(* Logix 5000 project; controller R1USB70001_CWRU_Scenario_Gen_20111116 vendor 1 type 14 code 54 rev 19.11; software revision 19.01; part 4 of 6 *)
(* tags used below, declared in another part *)
   EditScenarioPv : EditScenarioPv;
   HMIPv : HMIPv;
   CL_LP_B1_SG : ALIAS FOR ACNR_CP_SG_N5:1:O.1;
   CL_LP_ML_SG : ALIAS FOR ACNR_CP_SG_N5:1:O.0;
   EditScenario : EditScenarioPub;
   HMI : HMIPub;
   HMI_Intfc_Write_Buffer : DINT[20];
   RL_LP_B1_SG : ALIAS FOR ACNR_RP_SG_N4:1:O.1;
   RL_LP_B2_SG : ALIAS FOR ACNR_RP_SG_N4:2:O.4;
   RL_LP_B3_SG : ALIAS FOR ACNR_RP_SG_N4:3:O.7;
   RL_LP_B4_SG : ALIAS FOR ACNR_RP_SG_N4:5:O.2;
   RL_LP_ML_SG : ALIAS FOR ACNR_RP_SG_N4:1:O.0;
   Scenario : Scenario_Def[100];
(* MainProgram, continued *)

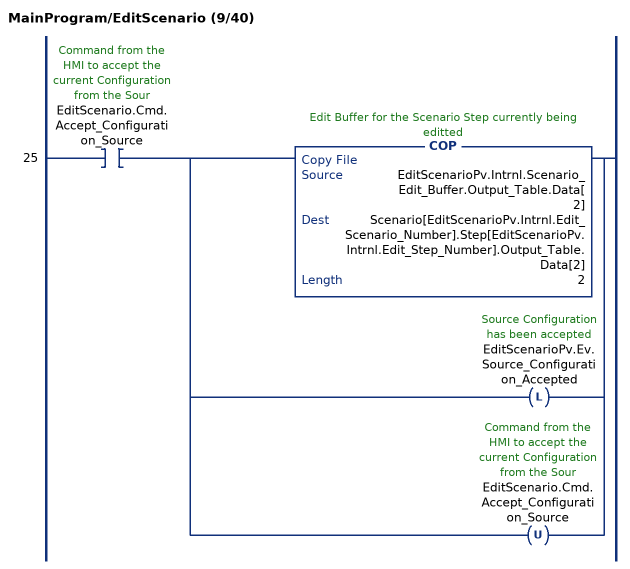
   25: XIC(EditScenario.Cmd.Accept_Configuration_Source)[COP(EditScenarioPv.Intrnl.Scenario_Edit_Buffer.Output_Table.Data[2],Scenario[EditScenarioPv.Intrnl.Edit_Scenario_Number].Step[EditScenarioPv.Intrnl.Edit_Step_Number].Output_Table.Data[2],2) ,OTL(EditScenarioPv.Ev.Source_Configuration_Accepted) ,OTU(EditScenario.Cmd.Accept_Configuration_Source) ];
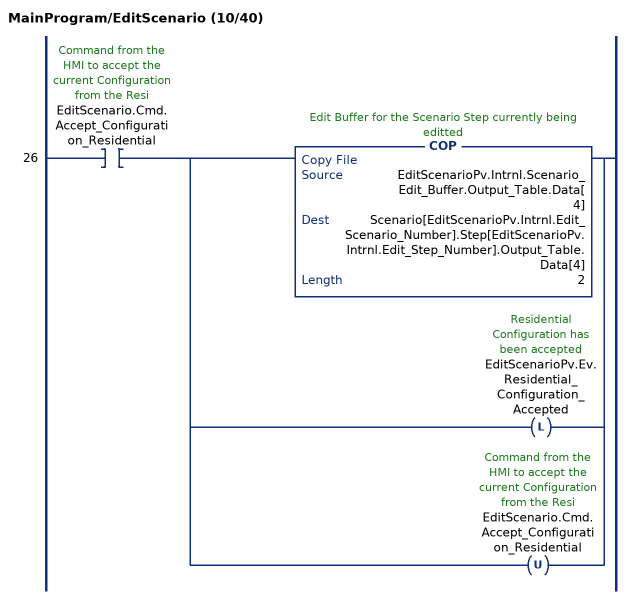
   26: XIC(EditScenario.Cmd.Accept_Configuration_Residential)[COP(EditScenarioPv.Intrnl.Scenario_Edit_Buffer.Output_Table.Data[4],Scenario[EditScenarioPv.Intrnl.Edit_Scenario_Number].Step[EditScenarioPv.Intrnl.Edit_Step_Number].Output_Table.Data[4],2) ,OTL(EditScenarioPv.Ev.Residential_Configuration_Accepted) ,OTU(EditScenario.Cmd.Accept_Configuration_Residential) ];
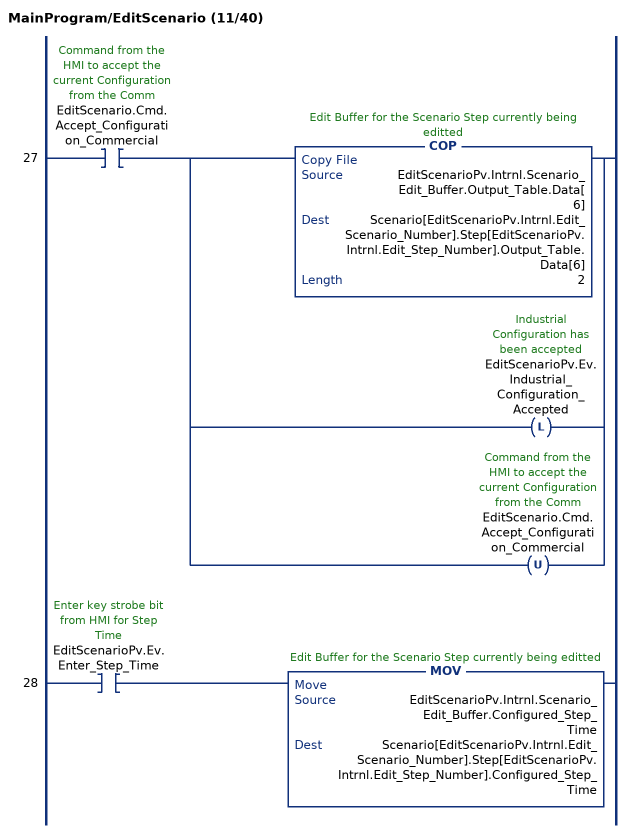
   27: XIC(EditScenario.Cmd.Accept_Configuration_Commercial)[COP(EditScenarioPv.Intrnl.Scenario_Edit_Buffer.Output_Table.Data[6],Scenario[EditScenarioPv.Intrnl.Edit_Scenario_Number].Step[EditScenarioPv.Intrnl.Edit_Step_Number].Output_Table.Data[6],2) ,OTL(EditScenarioPv.Ev.Industrial_Configuration_Accepted) ,OTU(EditScenario.Cmd.Accept_Configuration_Commercial) ];
   28: XIC(EditScenarioPv.Ev.Enter_Step_Time)MOV(EditScenarioPv.Intrnl.Scenario_Edit_Buffer.Configured_Step_Time,Scenario[EditScenarioPv.Intrnl.Edit_Scenario_Number].Step[EditScenarioPv.Intrnl.Edit_Step_Number].Configured_Step_Time);
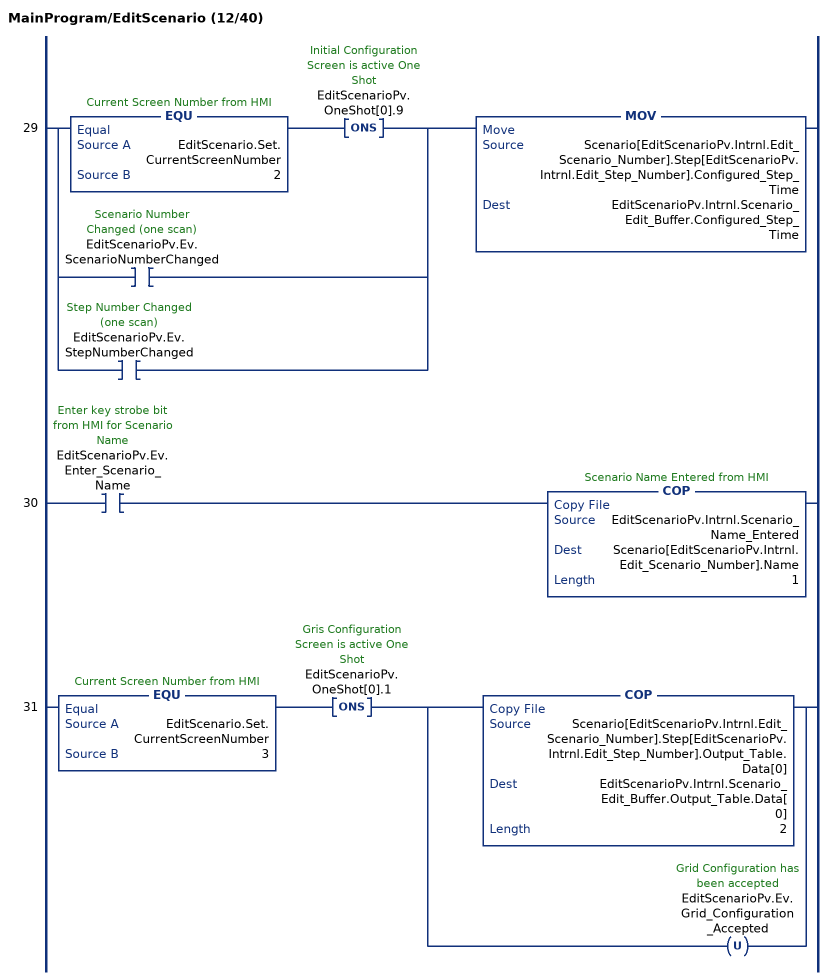
   29: [EQU(EditScenario.Set.CurrentScreenNumber,2) ONS(EditScenarioPv.OneShot[0].9) ,XIC(EditScenarioPv.Ev.ScenarioNumberChanged) ,XIC(EditScenarioPv.Ev.StepNumberChanged) ]MOV(Scenario[EditScenarioPv.Intrnl.Edit_Scenario_Number].Step[EditScenarioPv.Intrnl.Edit_Step_Number].Configured_Step_Time,EditScenarioPv.Intrnl.Scenario_Edit_Buffer.Configured_Step_Time);
   30: XIC(EditScenarioPv.Ev.Enter_Scenario_Name)COP(EditScenarioPv.Intrnl.Scenario_Name_Entered,Scenario[EditScenarioPv.Intrnl.Edit_Scenario_Number].Name,1);
   31: EQU(EditScenario.Set.CurrentScreenNumber,3)ONS(EditScenarioPv.OneShot[0].1)[COP(Scenario[EditScenarioPv.Intrnl.Edit_Scenario_Number].Step[EditScenarioPv.Intrnl.Edit_Step_Number].Output_Table.Data[0],EditScenarioPv.Intrnl.Scenario_Edit_Buffer.Output_Table.Data[0],2) ,OTU(EditScenarioPv.Ev.Grid_Configuration_Accepted) ];
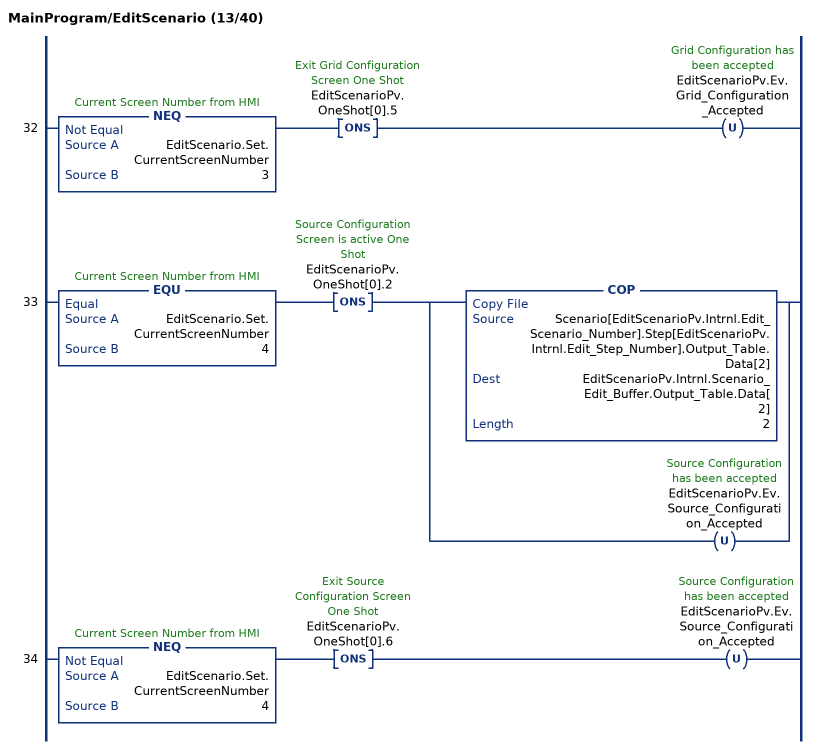
   32: NEQ(EditScenario.Set.CurrentScreenNumber,3)ONS(EditScenarioPv.OneShot[0].5)OTU(EditScenarioPv.Ev.Grid_Configuration_Accepted);
   33: EQU(EditScenario.Set.CurrentScreenNumber,4)ONS(EditScenarioPv.OneShot[0].2)[COP(Scenario[EditScenarioPv.Intrnl.Edit_Scenario_Number].Step[EditScenarioPv.Intrnl.Edit_Step_Number].Output_Table.Data[2],EditScenarioPv.Intrnl.Scenario_Edit_Buffer.Output_Table.Data[2],2) ,OTU(EditScenarioPv.Ev.Source_Configuration_Accepted) ];
   34: NEQ(EditScenario.Set.CurrentScreenNumber,4)ONS(EditScenarioPv.OneShot[0].6)OTU(EditScenarioPv.Ev.Source_Configuration_Accepted);
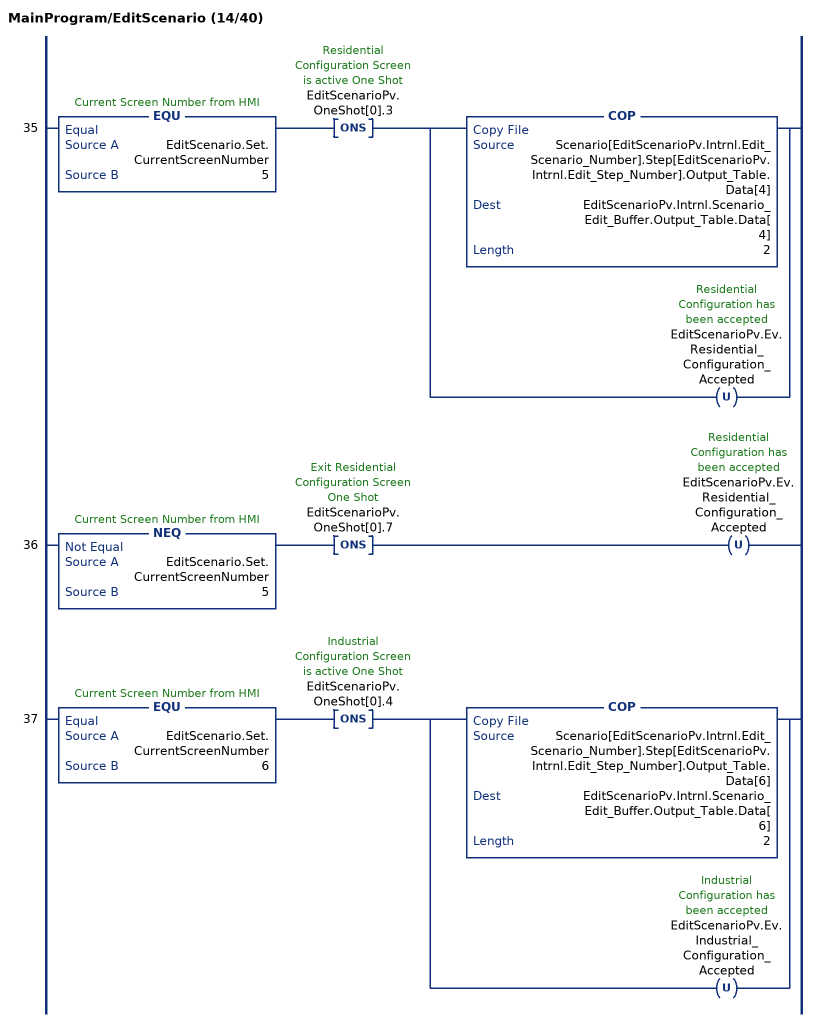
   35: EQU(EditScenario.Set.CurrentScreenNumber,5)ONS(EditScenarioPv.OneShot[0].3)[COP(Scenario[EditScenarioPv.Intrnl.Edit_Scenario_Number].Step[EditScenarioPv.Intrnl.Edit_Step_Number].Output_Table.Data[4],EditScenarioPv.Intrnl.Scenario_Edit_Buffer.Output_Table.Data[4],2) ,OTU(EditScenarioPv.Ev.Residential_Configuration_Accepted) ];
   36: NEQ(EditScenario.Set.CurrentScreenNumber,5)ONS(EditScenarioPv.OneShot[0].7)OTU(EditScenarioPv.Ev.Residential_Configuration_Accepted);
   37: EQU(EditScenario.Set.CurrentScreenNumber,6)ONS(EditScenarioPv.OneShot[0].4)[COP(Scenario[EditScenarioPv.Intrnl.Edit_Scenario_Number].Step[EditScenarioPv.Intrnl.Edit_Step_Number].Output_Table.Data[6],EditScenarioPv.Intrnl.Scenario_Edit_Buffer.Output_Table.Data[6],2) ,OTU(EditScenarioPv.Ev.Industrial_Configuration_Accepted) ];
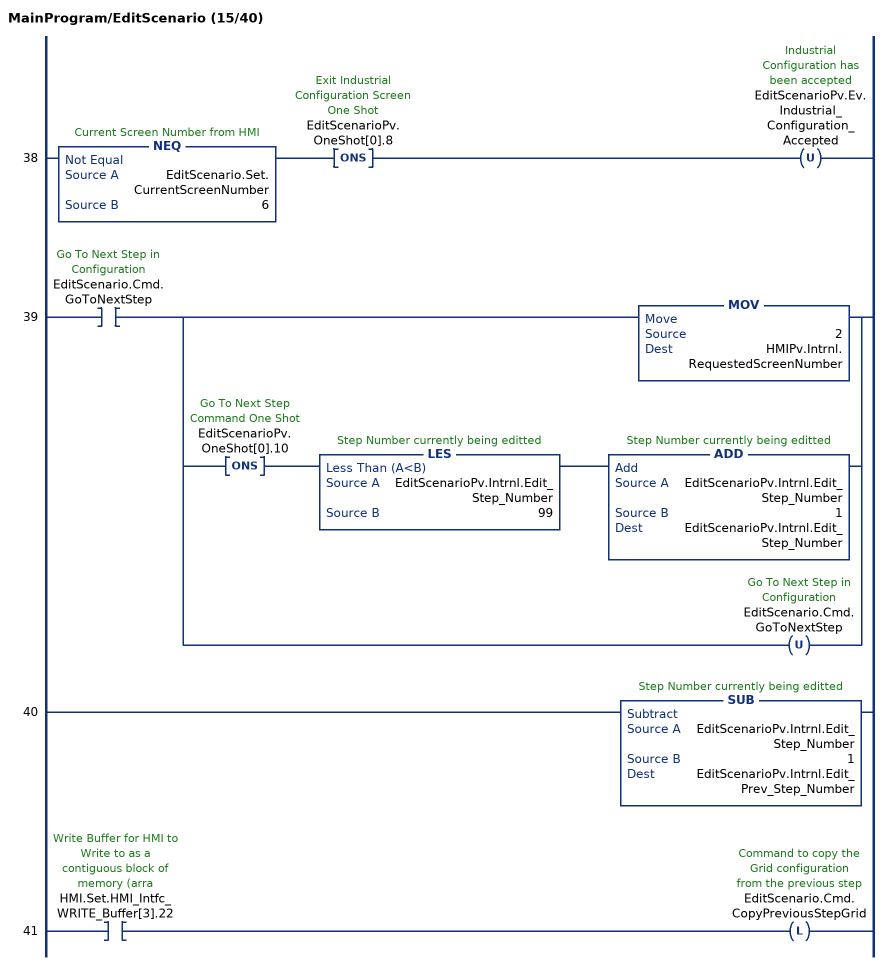
   38: NEQ(EditScenario.Set.CurrentScreenNumber,6)ONS(EditScenarioPv.OneShot[0].8)OTU(EditScenarioPv.Ev.Industrial_Configuration_Accepted);
   39: XIC(EditScenario.Cmd.GoToNextStep)[MOV(2,HMIPv.Intrnl.RequestedScreenNumber) ,ONS(EditScenarioPv.OneShot[0].10) LES(EditScenarioPv.Intrnl.Edit_Step_Number,99) ADD(EditScenarioPv.Intrnl.Edit_Step_Number,1,EditScenarioPv.Intrnl.Edit_Step_Number) ,OTU(EditScenario.Cmd.GoToNextStep) ];
   40: SUB(EditScenarioPv.Intrnl.Edit_Step_Number,1,EditScenarioPv.Intrnl.Edit_Prev_Step_Number);
   41: XIC(HMI.Set.HMI_Intfc_WRITE_Buffer[3].22)OTL(EditScenario.Cmd.CopyPreviousStepGrid);
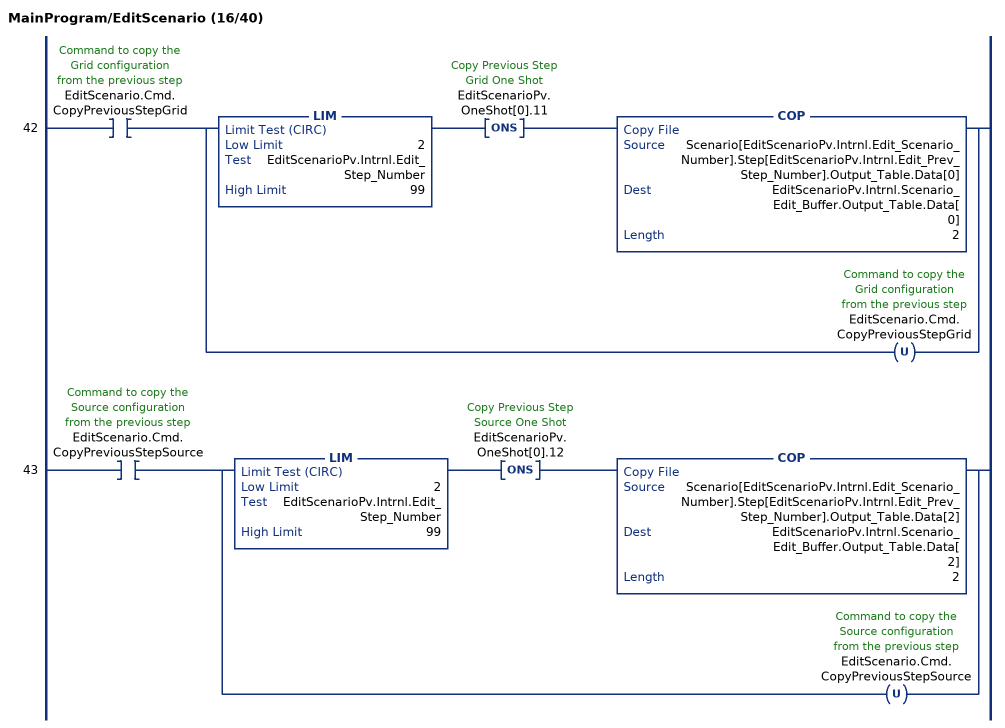
   42: XIC(EditScenario.Cmd.CopyPreviousStepGrid)[LIM(2,EditScenarioPv.Intrnl.Edit_Step_Number,99) ONS(EditScenarioPv.OneShot[0].11) COP(Scenario[EditScenarioPv.Intrnl.Edit_Scenario_Number].Step[EditScenarioPv.Intrnl.Edit_Prev_Step_Number].Output_Table.Data[0],EditScenarioPv.Intrnl.Scenario_Edit_Buffer.Output_Table.Data[0],2) ,OTU(EditScenario.Cmd.CopyPreviousStepGrid) ];
   43: XIC(EditScenario.Cmd.CopyPreviousStepSource)[LIM(2,EditScenarioPv.Intrnl.Edit_Step_Number,99) ONS(EditScenarioPv.OneShot[0].12) COP(Scenario[EditScenarioPv.Intrnl.Edit_Scenario_Number].Step[EditScenarioPv.Intrnl.Edit_Prev_Step_Number].Output_Table.Data[2],EditScenarioPv.Intrnl.Scenario_Edit_Buffer.Output_Table.Data[2],2) ,OTU(EditScenario.Cmd.CopyPreviousStepSource) ];
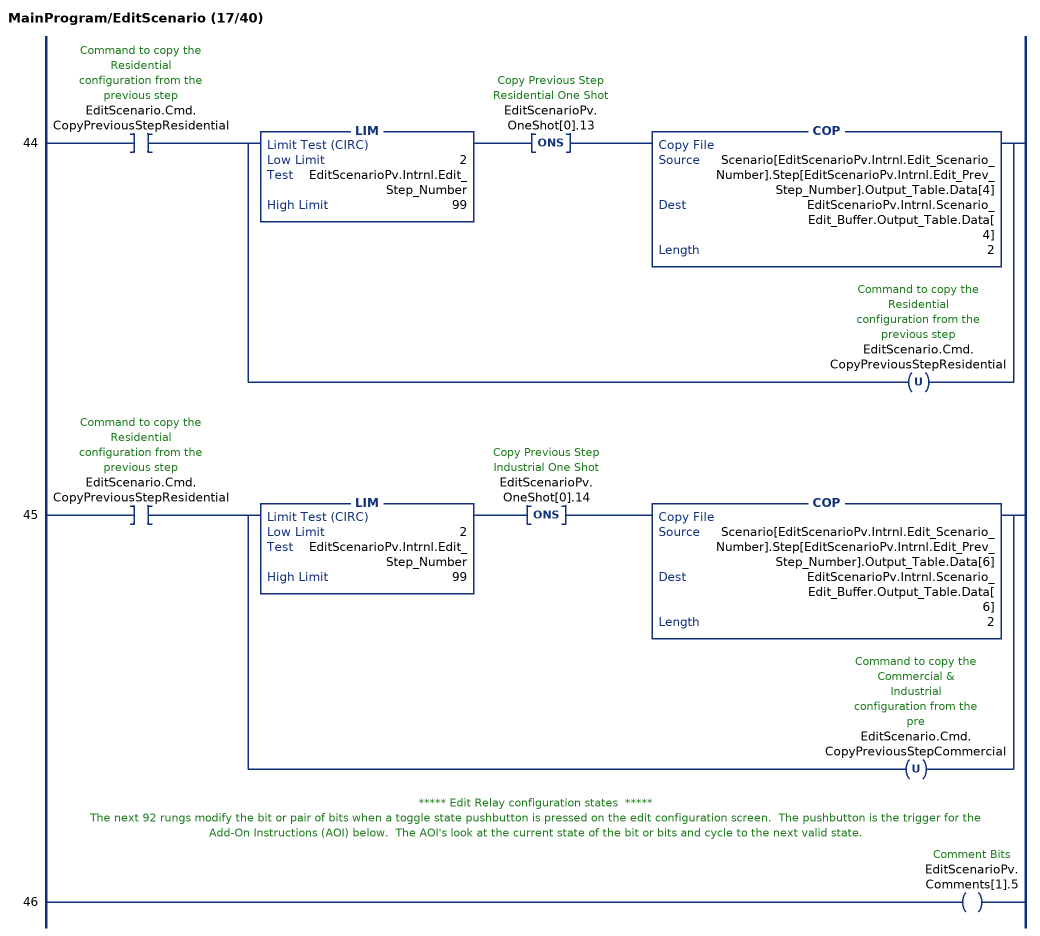
   44: XIC(EditScenario.Cmd.CopyPreviousStepResidential)[LIM(2,EditScenarioPv.Intrnl.Edit_Step_Number,99) ONS(EditScenarioPv.OneShot[0].13) COP(Scenario[EditScenarioPv.Intrnl.Edit_Scenario_Number].Step[EditScenarioPv.Intrnl.Edit_Prev_Step_Number].Output_Table.Data[4],EditScenarioPv.Intrnl.Scenario_Edit_Buffer.Output_Table.Data[4],2) ,OTU(EditScenario.Cmd.CopyPreviousStepResidential) ];
   45: XIC(EditScenario.Cmd.CopyPreviousStepResidential)[LIM(2,EditScenarioPv.Intrnl.Edit_Step_Number,99) ONS(EditScenarioPv.OneShot[0].14) COP(Scenario[EditScenarioPv.Intrnl.Edit_Scenario_Number].Step[EditScenarioPv.Intrnl.Edit_Prev_Step_Number].Output_Table.Data[6],EditScenarioPv.Intrnl.Scenario_Edit_Buffer.Output_Table.Data[6],2) ,OTU(EditScenario.Cmd.CopyPreviousStepCommercial) ];
   // ***** Edit Relay configuration states  *****
   // The next 92 rungs modify the bit or pair of bits when a toggle state pushbutton is pressed on the edit configuration screen.  The pushbutton is the trigger for the Add-On Instructions (AOI) below.  The AOI's look at the current state of the bit or bits and cycle to the next valid state.
   46: OTE(EditScenarioPv.Comments[1].5);
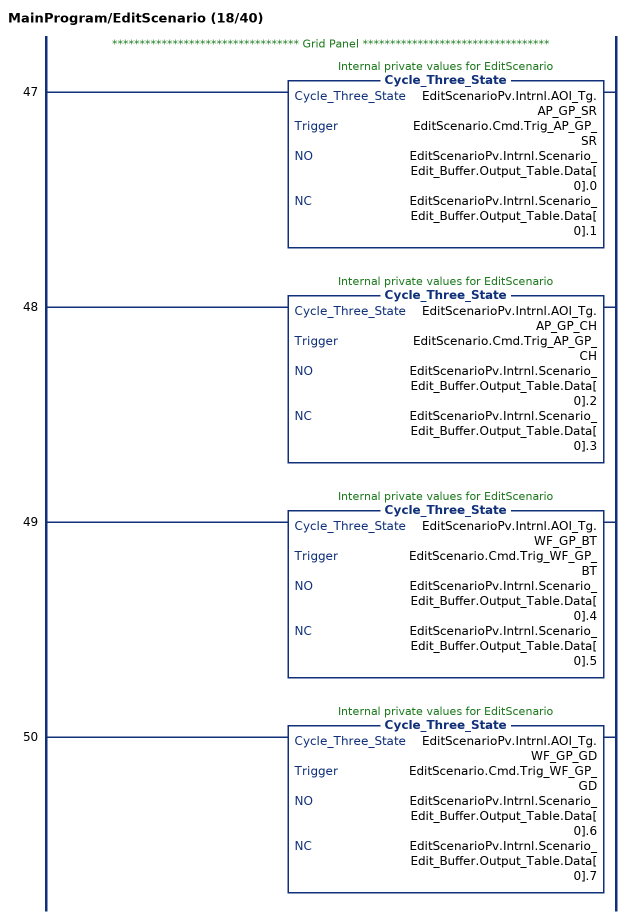
   // ********************************** Grid Panel **********************************
   47: Cycle_Three_State(EditScenarioPv.Intrnl.AOI_Tg.AP_GP_SR,EditScenario.Cmd.Trig_AP_GP_SR,EditScenarioPv.Intrnl.Scenario_Edit_Buffer.Output_Table.Data[0].0,EditScenarioPv.Intrnl.Scenario_Edit_Buffer.Output_Table.Data[0].1);
   48: Cycle_Three_State(EditScenarioPv.Intrnl.AOI_Tg.AP_GP_CH,EditScenario.Cmd.Trig_AP_GP_CH,EditScenarioPv.Intrnl.Scenario_Edit_Buffer.Output_Table.Data[0].2,EditScenarioPv.Intrnl.Scenario_Edit_Buffer.Output_Table.Data[0].3);
   49: Cycle_Three_State(EditScenarioPv.Intrnl.AOI_Tg.WF_GP_BT,EditScenario.Cmd.Trig_WF_GP_BT,EditScenarioPv.Intrnl.Scenario_Edit_Buffer.Output_Table.Data[0].4,EditScenarioPv.Intrnl.Scenario_Edit_Buffer.Output_Table.Data[0].5);
   50: Cycle_Three_State(EditScenarioPv.Intrnl.AOI_Tg.WF_GP_GD,EditScenario.Cmd.Trig_WF_GP_GD,EditScenarioPv.Intrnl.Scenario_Edit_Buffer.Output_Table.Data[0].6,EditScenarioPv.Intrnl.Scenario_Edit_Buffer.Output_Table.Data[0].7);
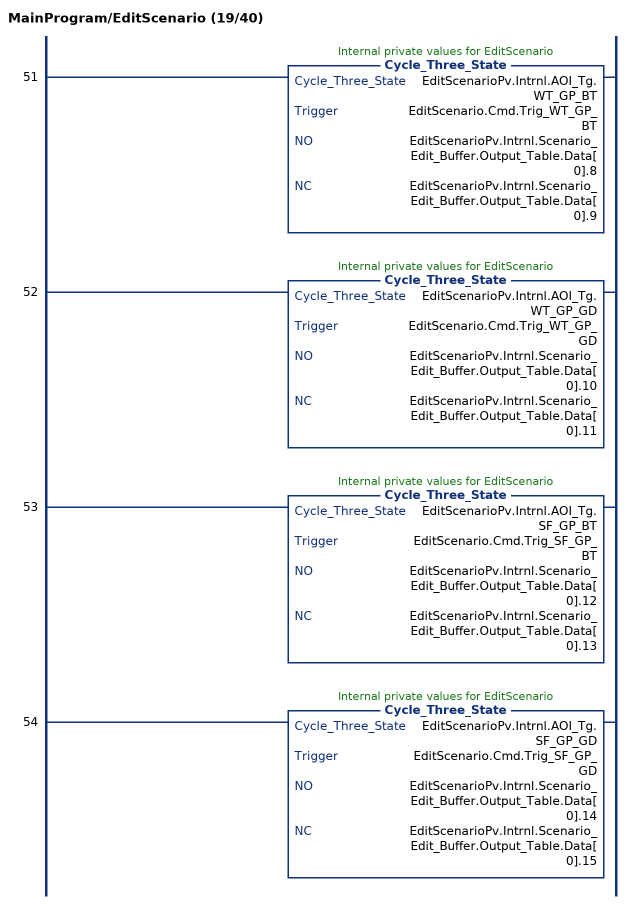
   51: Cycle_Three_State(EditScenarioPv.Intrnl.AOI_Tg.WT_GP_BT,EditScenario.Cmd.Trig_WT_GP_BT,EditScenarioPv.Intrnl.Scenario_Edit_Buffer.Output_Table.Data[0].8,EditScenarioPv.Intrnl.Scenario_Edit_Buffer.Output_Table.Data[0].9);
   52: Cycle_Three_State(EditScenarioPv.Intrnl.AOI_Tg.WT_GP_GD,EditScenario.Cmd.Trig_WT_GP_GD,EditScenarioPv.Intrnl.Scenario_Edit_Buffer.Output_Table.Data[0].10,EditScenarioPv.Intrnl.Scenario_Edit_Buffer.Output_Table.Data[0].11);
   53: Cycle_Three_State(EditScenarioPv.Intrnl.AOI_Tg.SF_GP_BT,EditScenario.Cmd.Trig_SF_GP_BT,EditScenarioPv.Intrnl.Scenario_Edit_Buffer.Output_Table.Data[0].12,EditScenarioPv.Intrnl.Scenario_Edit_Buffer.Output_Table.Data[0].13);
   54: Cycle_Three_State(EditScenarioPv.Intrnl.AOI_Tg.SF_GP_GD,EditScenario.Cmd.Trig_SF_GP_GD,EditScenarioPv.Intrnl.Scenario_Edit_Buffer.Output_Table.Data[0].14,EditScenarioPv.Intrnl.Scenario_Edit_Buffer.Output_Table.Data[0].15);
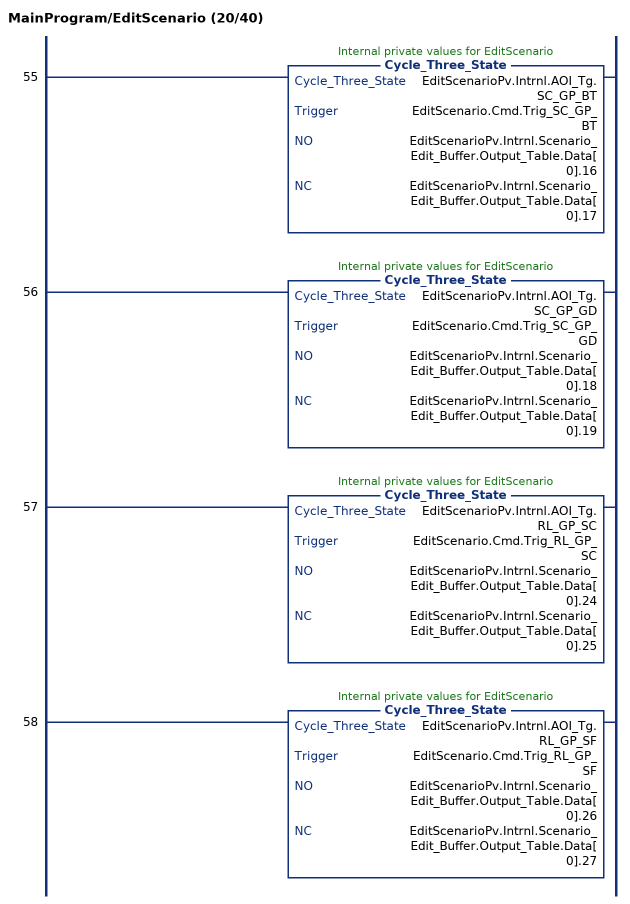
   55: Cycle_Three_State(EditScenarioPv.Intrnl.AOI_Tg.SC_GP_BT,EditScenario.Cmd.Trig_SC_GP_BT,EditScenarioPv.Intrnl.Scenario_Edit_Buffer.Output_Table.Data[0].16,EditScenarioPv.Intrnl.Scenario_Edit_Buffer.Output_Table.Data[0].17);
   56: Cycle_Three_State(EditScenarioPv.Intrnl.AOI_Tg.SC_GP_GD,EditScenario.Cmd.Trig_SC_GP_GD,EditScenarioPv.Intrnl.Scenario_Edit_Buffer.Output_Table.Data[0].18,EditScenarioPv.Intrnl.Scenario_Edit_Buffer.Output_Table.Data[0].19);
   57: Cycle_Three_State(EditScenarioPv.Intrnl.AOI_Tg.RL_GP_SC,EditScenario.Cmd.Trig_RL_GP_SC,EditScenarioPv.Intrnl.Scenario_Edit_Buffer.Output_Table.Data[0].24,EditScenarioPv.Intrnl.Scenario_Edit_Buffer.Output_Table.Data[0].25);
   58: Cycle_Three_State(EditScenarioPv.Intrnl.AOI_Tg.RL_GP_SF,EditScenario.Cmd.Trig_RL_GP_SF,EditScenarioPv.Intrnl.Scenario_Edit_Buffer.Output_Table.Data[0].26,EditScenarioPv.Intrnl.Scenario_Edit_Buffer.Output_Table.Data[0].27);
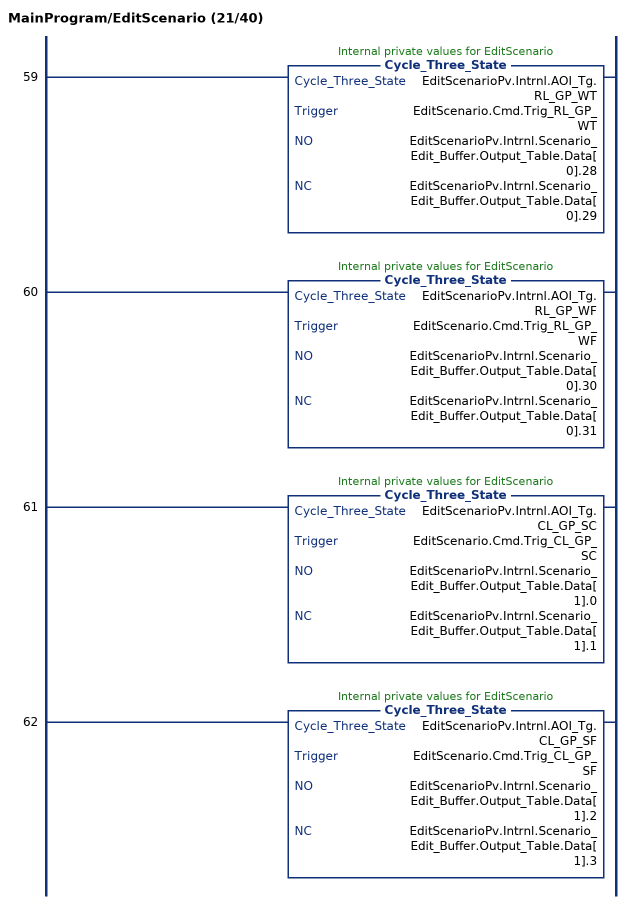
   59: Cycle_Three_State(EditScenarioPv.Intrnl.AOI_Tg.RL_GP_WT,EditScenario.Cmd.Trig_RL_GP_WT,EditScenarioPv.Intrnl.Scenario_Edit_Buffer.Output_Table.Data[0].28,EditScenarioPv.Intrnl.Scenario_Edit_Buffer.Output_Table.Data[0].29);
   60: Cycle_Three_State(EditScenarioPv.Intrnl.AOI_Tg.RL_GP_WF,EditScenario.Cmd.Trig_RL_GP_WF,EditScenarioPv.Intrnl.Scenario_Edit_Buffer.Output_Table.Data[0].30,EditScenarioPv.Intrnl.Scenario_Edit_Buffer.Output_Table.Data[0].31);
   61: Cycle_Three_State(EditScenarioPv.Intrnl.AOI_Tg.CL_GP_SC,EditScenario.Cmd.Trig_CL_GP_SC,EditScenarioPv.Intrnl.Scenario_Edit_Buffer.Output_Table.Data[1].0,EditScenarioPv.Intrnl.Scenario_Edit_Buffer.Output_Table.Data[1].1);
   62: Cycle_Three_State(EditScenarioPv.Intrnl.AOI_Tg.CL_GP_SF,EditScenario.Cmd.Trig_CL_GP_SF,EditScenarioPv.Intrnl.Scenario_Edit_Buffer.Output_Table.Data[1].2,EditScenarioPv.Intrnl.Scenario_Edit_Buffer.Output_Table.Data[1].3);
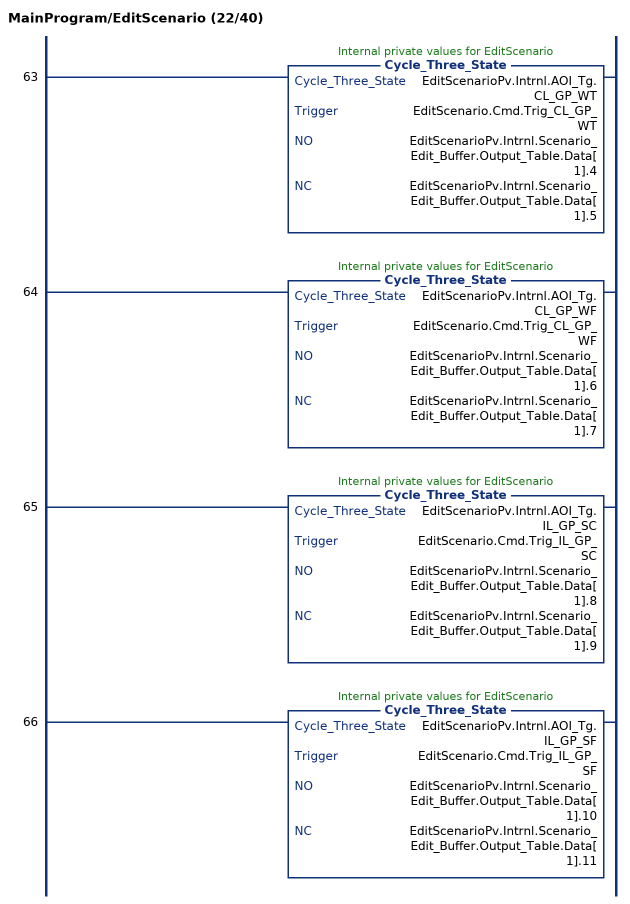
   63: Cycle_Three_State(EditScenarioPv.Intrnl.AOI_Tg.CL_GP_WT,EditScenario.Cmd.Trig_CL_GP_WT,EditScenarioPv.Intrnl.Scenario_Edit_Buffer.Output_Table.Data[1].4,EditScenarioPv.Intrnl.Scenario_Edit_Buffer.Output_Table.Data[1].5);
   64: Cycle_Three_State(EditScenarioPv.Intrnl.AOI_Tg.CL_GP_WF,EditScenario.Cmd.Trig_CL_GP_WF,EditScenarioPv.Intrnl.Scenario_Edit_Buffer.Output_Table.Data[1].6,EditScenarioPv.Intrnl.Scenario_Edit_Buffer.Output_Table.Data[1].7);
   65: Cycle_Three_State(EditScenarioPv.Intrnl.AOI_Tg.IL_GP_SC,EditScenario.Cmd.Trig_IL_GP_SC,EditScenarioPv.Intrnl.Scenario_Edit_Buffer.Output_Table.Data[1].8,EditScenarioPv.Intrnl.Scenario_Edit_Buffer.Output_Table.Data[1].9);
   66: Cycle_Three_State(EditScenarioPv.Intrnl.AOI_Tg.IL_GP_SF,EditScenario.Cmd.Trig_IL_GP_SF,EditScenarioPv.Intrnl.Scenario_Edit_Buffer.Output_Table.Data[1].10,EditScenarioPv.Intrnl.Scenario_Edit_Buffer.Output_Table.Data[1].11);
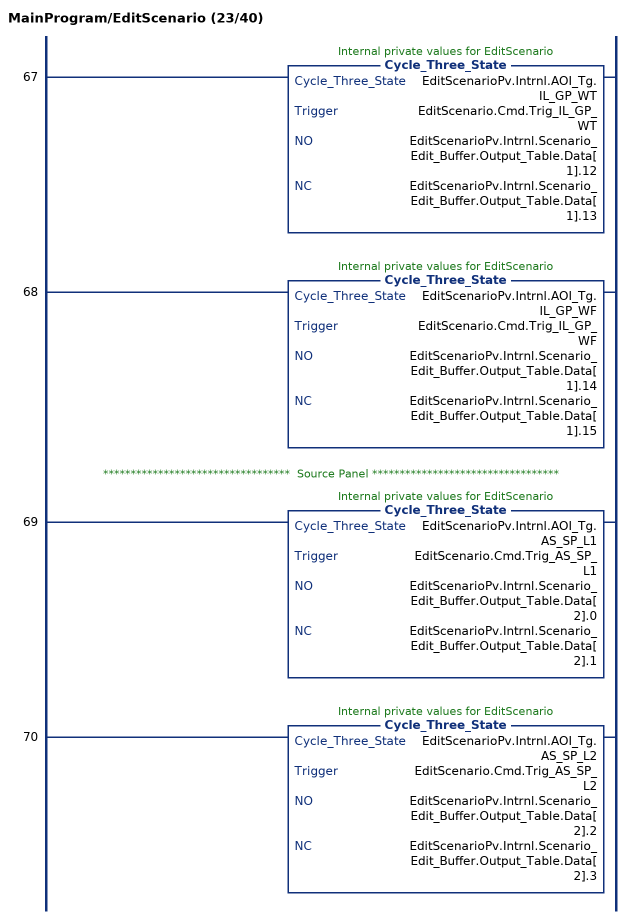
   67: Cycle_Three_State(EditScenarioPv.Intrnl.AOI_Tg.IL_GP_WT,EditScenario.Cmd.Trig_IL_GP_WT,EditScenarioPv.Intrnl.Scenario_Edit_Buffer.Output_Table.Data[1].12,EditScenarioPv.Intrnl.Scenario_Edit_Buffer.Output_Table.Data[1].13);
   68: Cycle_Three_State(EditScenarioPv.Intrnl.AOI_Tg.IL_GP_WF,EditScenario.Cmd.Trig_IL_GP_WF,EditScenarioPv.Intrnl.Scenario_Edit_Buffer.Output_Table.Data[1].14,EditScenarioPv.Intrnl.Scenario_Edit_Buffer.Output_Table.Data[1].15);
   // **********************************  Source Panel **********************************
   69: Cycle_Three_State(EditScenarioPv.Intrnl.AOI_Tg.AS_SP_L1,EditScenario.Cmd.Trig_AS_SP_L1,EditScenarioPv.Intrnl.Scenario_Edit_Buffer.Output_Table.Data[2].0,EditScenarioPv.Intrnl.Scenario_Edit_Buffer.Output_Table.Data[2].1);
   70: Cycle_Three_State(EditScenarioPv.Intrnl.AOI_Tg.AS_SP_L2,EditScenario.Cmd.Trig_AS_SP_L2,EditScenarioPv.Intrnl.Scenario_Edit_Buffer.Output_Table.Data[2].2,EditScenarioPv.Intrnl.Scenario_Edit_Buffer.Output_Table.Data[2].3);
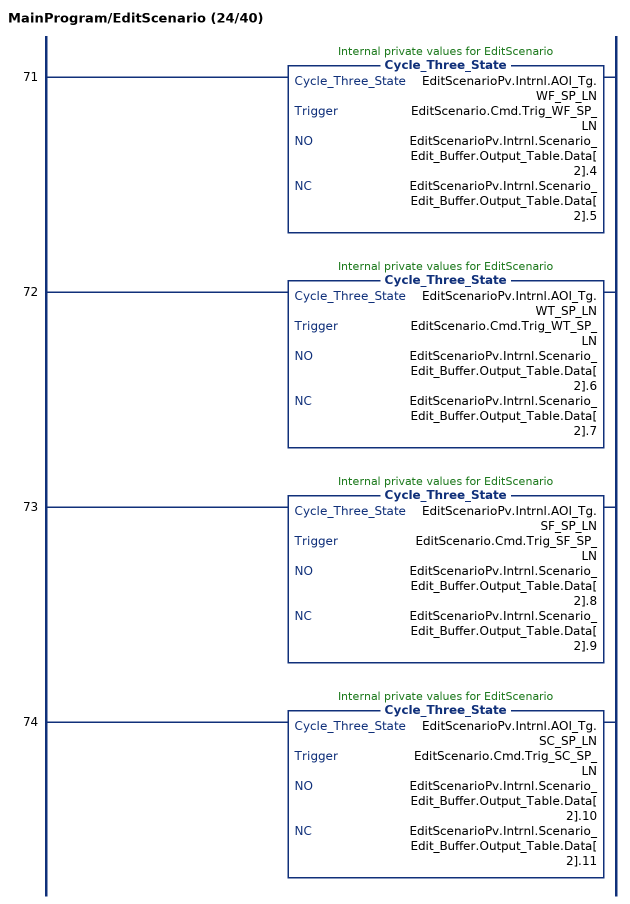
   71: Cycle_Three_State(EditScenarioPv.Intrnl.AOI_Tg.WF_SP_LN,EditScenario.Cmd.Trig_WF_SP_LN,EditScenarioPv.Intrnl.Scenario_Edit_Buffer.Output_Table.Data[2].4,EditScenarioPv.Intrnl.Scenario_Edit_Buffer.Output_Table.Data[2].5);
   72: Cycle_Three_State(EditScenarioPv.Intrnl.AOI_Tg.WT_SP_LN,EditScenario.Cmd.Trig_WT_SP_LN,EditScenarioPv.Intrnl.Scenario_Edit_Buffer.Output_Table.Data[2].6,EditScenarioPv.Intrnl.Scenario_Edit_Buffer.Output_Table.Data[2].7);
   73: Cycle_Three_State(EditScenarioPv.Intrnl.AOI_Tg.SF_SP_LN,EditScenario.Cmd.Trig_SF_SP_LN,EditScenarioPv.Intrnl.Scenario_Edit_Buffer.Output_Table.Data[2].8,EditScenarioPv.Intrnl.Scenario_Edit_Buffer.Output_Table.Data[2].9);
   74: Cycle_Three_State(EditScenarioPv.Intrnl.AOI_Tg.SC_SP_LN,EditScenario.Cmd.Trig_SC_SP_LN,EditScenarioPv.Intrnl.Scenario_Edit_Buffer.Output_Table.Data[2].10,EditScenarioPv.Intrnl.Scenario_Edit_Buffer.Output_Table.Data[2].11);
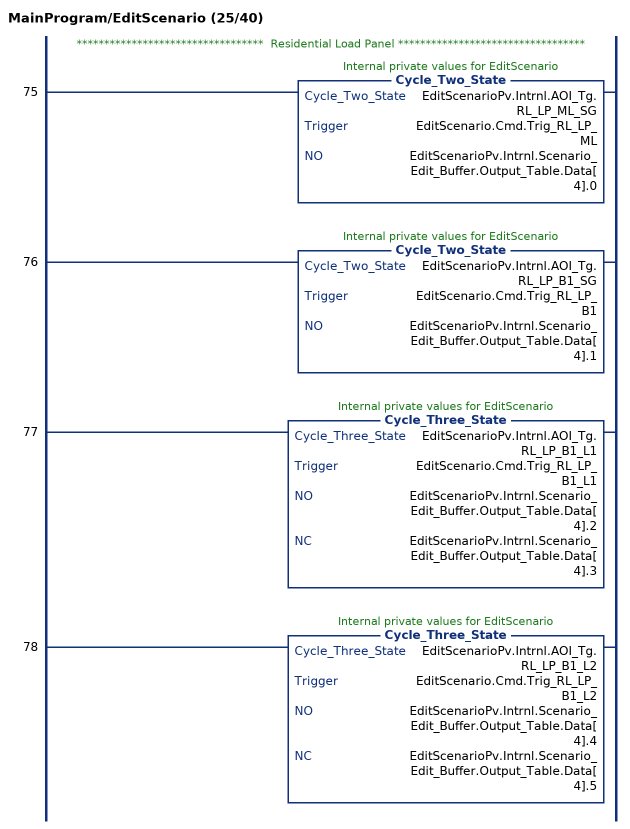
   // **********************************  Residential Load Panel **********************************
   75: Cycle_Two_State(EditScenarioPv.Intrnl.AOI_Tg.RL_LP_ML_SG,EditScenario.Cmd.Trig_RL_LP_ML,EditScenarioPv.Intrnl.Scenario_Edit_Buffer.Output_Table.Data[4].0);
   76: Cycle_Two_State(EditScenarioPv.Intrnl.AOI_Tg.RL_LP_B1_SG,EditScenario.Cmd.Trig_RL_LP_B1,EditScenarioPv.Intrnl.Scenario_Edit_Buffer.Output_Table.Data[4].1);
   77: Cycle_Three_State(EditScenarioPv.Intrnl.AOI_Tg.RL_LP_B1_L1,EditScenario.Cmd.Trig_RL_LP_B1_L1,EditScenarioPv.Intrnl.Scenario_Edit_Buffer.Output_Table.Data[4].2,EditScenarioPv.Intrnl.Scenario_Edit_Buffer.Output_Table.Data[4].3);
   78: Cycle_Three_State(EditScenarioPv.Intrnl.AOI_Tg.RL_LP_B1_L2,EditScenario.Cmd.Trig_RL_LP_B1_L2,EditScenarioPv.Intrnl.Scenario_Edit_Buffer.Output_Table.Data[4].4,EditScenarioPv.Intrnl.Scenario_Edit_Buffer.Output_Table.Data[4].5);
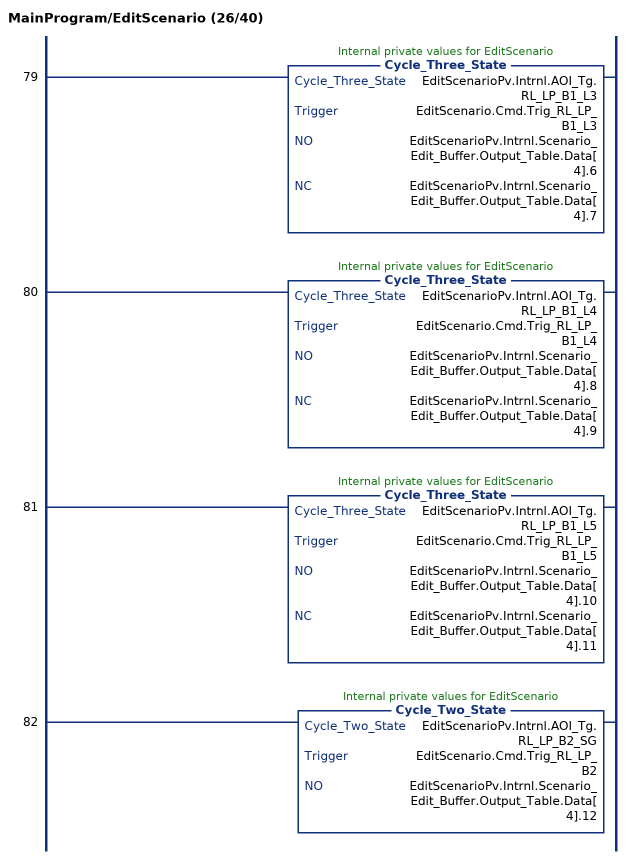
   79: Cycle_Three_State(EditScenarioPv.Intrnl.AOI_Tg.RL_LP_B1_L3,EditScenario.Cmd.Trig_RL_LP_B1_L3,EditScenarioPv.Intrnl.Scenario_Edit_Buffer.Output_Table.Data[4].6,EditScenarioPv.Intrnl.Scenario_Edit_Buffer.Output_Table.Data[4].7);
   80: Cycle_Three_State(EditScenarioPv.Intrnl.AOI_Tg.RL_LP_B1_L4,EditScenario.Cmd.Trig_RL_LP_B1_L4,EditScenarioPv.Intrnl.Scenario_Edit_Buffer.Output_Table.Data[4].8,EditScenarioPv.Intrnl.Scenario_Edit_Buffer.Output_Table.Data[4].9);
   81: Cycle_Three_State(EditScenarioPv.Intrnl.AOI_Tg.RL_LP_B1_L5,EditScenario.Cmd.Trig_RL_LP_B1_L5,EditScenarioPv.Intrnl.Scenario_Edit_Buffer.Output_Table.Data[4].10,EditScenarioPv.Intrnl.Scenario_Edit_Buffer.Output_Table.Data[4].11);
   82: Cycle_Two_State(EditScenarioPv.Intrnl.AOI_Tg.RL_LP_B2_SG,EditScenario.Cmd.Trig_RL_LP_B2,EditScenarioPv.Intrnl.Scenario_Edit_Buffer.Output_Table.Data[4].12);
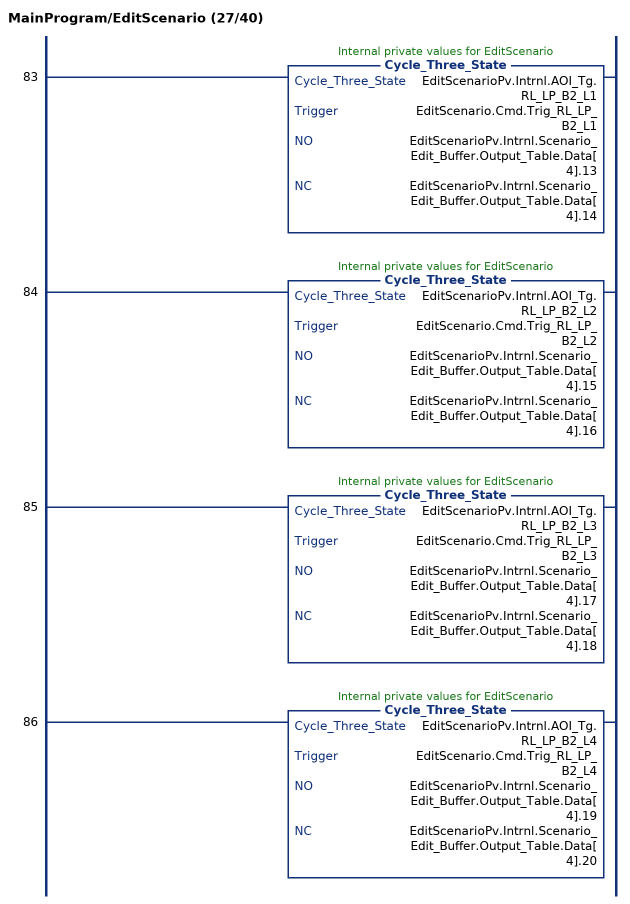
   83: Cycle_Three_State(EditScenarioPv.Intrnl.AOI_Tg.RL_LP_B2_L1,EditScenario.Cmd.Trig_RL_LP_B2_L1,EditScenarioPv.Intrnl.Scenario_Edit_Buffer.Output_Table.Data[4].13,EditScenarioPv.Intrnl.Scenario_Edit_Buffer.Output_Table.Data[4].14);
   84: Cycle_Three_State(EditScenarioPv.Intrnl.AOI_Tg.RL_LP_B2_L2,EditScenario.Cmd.Trig_RL_LP_B2_L2,EditScenarioPv.Intrnl.Scenario_Edit_Buffer.Output_Table.Data[4].15,EditScenarioPv.Intrnl.Scenario_Edit_Buffer.Output_Table.Data[4].16);
   85: Cycle_Three_State(EditScenarioPv.Intrnl.AOI_Tg.RL_LP_B2_L3,EditScenario.Cmd.Trig_RL_LP_B2_L3,EditScenarioPv.Intrnl.Scenario_Edit_Buffer.Output_Table.Data[4].17,EditScenarioPv.Intrnl.Scenario_Edit_Buffer.Output_Table.Data[4].18);
   86: Cycle_Three_State(EditScenarioPv.Intrnl.AOI_Tg.RL_LP_B2_L4,EditScenario.Cmd.Trig_RL_LP_B2_L4,EditScenarioPv.Intrnl.Scenario_Edit_Buffer.Output_Table.Data[4].19,EditScenarioPv.Intrnl.Scenario_Edit_Buffer.Output_Table.Data[4].20);
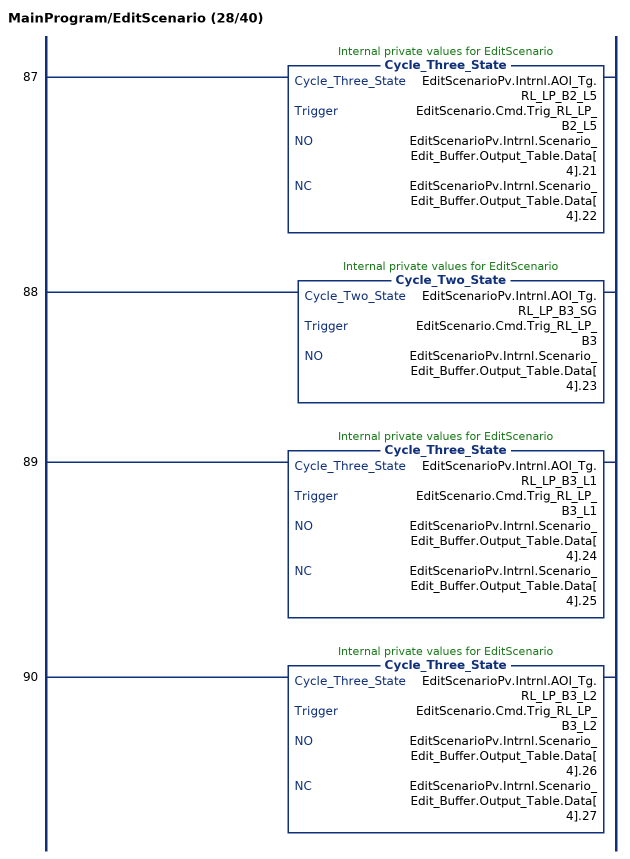
   87: Cycle_Three_State(EditScenarioPv.Intrnl.AOI_Tg.RL_LP_B2_L5,EditScenario.Cmd.Trig_RL_LP_B2_L5,EditScenarioPv.Intrnl.Scenario_Edit_Buffer.Output_Table.Data[4].21,EditScenarioPv.Intrnl.Scenario_Edit_Buffer.Output_Table.Data[4].22);
   88: Cycle_Two_State(EditScenarioPv.Intrnl.AOI_Tg.RL_LP_B3_SG,EditScenario.Cmd.Trig_RL_LP_B3,EditScenarioPv.Intrnl.Scenario_Edit_Buffer.Output_Table.Data[4].23);
   89: Cycle_Three_State(EditScenarioPv.Intrnl.AOI_Tg.RL_LP_B3_L1,EditScenario.Cmd.Trig_RL_LP_B3_L1,EditScenarioPv.Intrnl.Scenario_Edit_Buffer.Output_Table.Data[4].24,EditScenarioPv.Intrnl.Scenario_Edit_Buffer.Output_Table.Data[4].25);
   90: Cycle_Three_State(EditScenarioPv.Intrnl.AOI_Tg.RL_LP_B3_L2,EditScenario.Cmd.Trig_RL_LP_B3_L2,EditScenarioPv.Intrnl.Scenario_Edit_Buffer.Output_Table.Data[4].26,EditScenarioPv.Intrnl.Scenario_Edit_Buffer.Output_Table.Data[4].27);
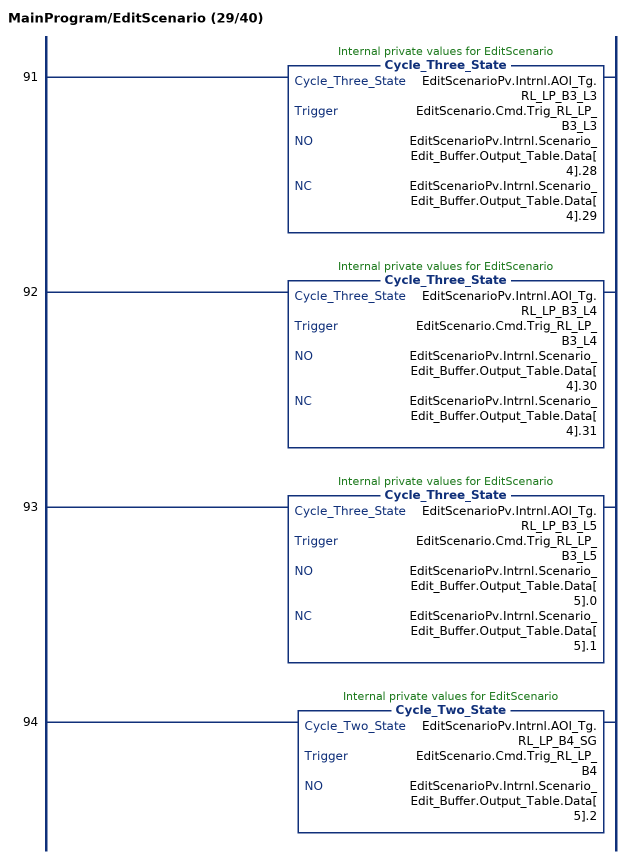
   91: Cycle_Three_State(EditScenarioPv.Intrnl.AOI_Tg.RL_LP_B3_L3,EditScenario.Cmd.Trig_RL_LP_B3_L3,EditScenarioPv.Intrnl.Scenario_Edit_Buffer.Output_Table.Data[4].28,EditScenarioPv.Intrnl.Scenario_Edit_Buffer.Output_Table.Data[4].29);
   92: Cycle_Three_State(EditScenarioPv.Intrnl.AOI_Tg.RL_LP_B3_L4,EditScenario.Cmd.Trig_RL_LP_B3_L4,EditScenarioPv.Intrnl.Scenario_Edit_Buffer.Output_Table.Data[4].30,EditScenarioPv.Intrnl.Scenario_Edit_Buffer.Output_Table.Data[4].31);
   93: Cycle_Three_State(EditScenarioPv.Intrnl.AOI_Tg.RL_LP_B3_L5,EditScenario.Cmd.Trig_RL_LP_B3_L5,EditScenarioPv.Intrnl.Scenario_Edit_Buffer.Output_Table.Data[5].0,EditScenarioPv.Intrnl.Scenario_Edit_Buffer.Output_Table.Data[5].1);
   94: Cycle_Two_State(EditScenarioPv.Intrnl.AOI_Tg.RL_LP_B4_SG,EditScenario.Cmd.Trig_RL_LP_B4,EditScenarioPv.Intrnl.Scenario_Edit_Buffer.Output_Table.Data[5].2);
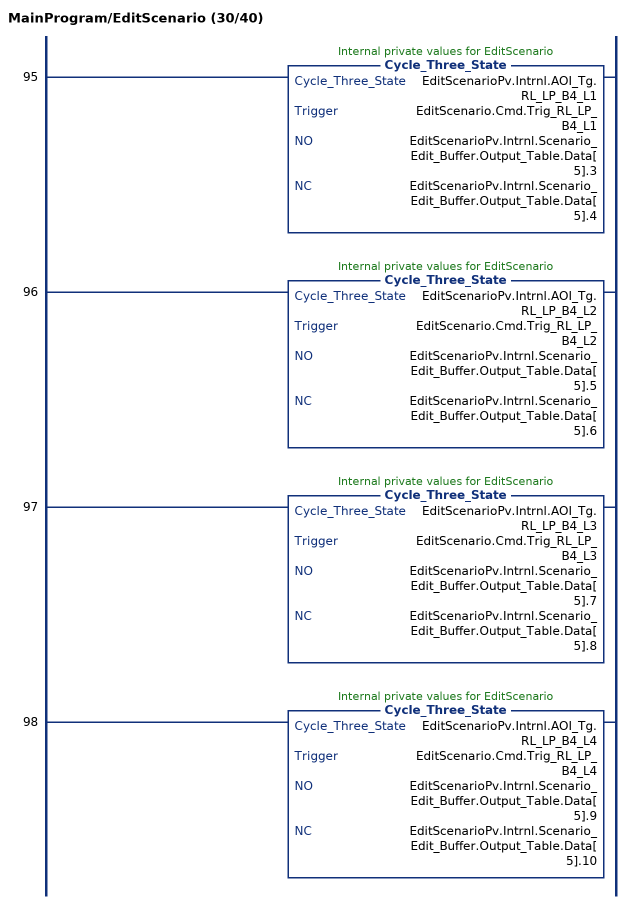
   95: Cycle_Three_State(EditScenarioPv.Intrnl.AOI_Tg.RL_LP_B4_L1,EditScenario.Cmd.Trig_RL_LP_B4_L1,EditScenarioPv.Intrnl.Scenario_Edit_Buffer.Output_Table.Data[5].3,EditScenarioPv.Intrnl.Scenario_Edit_Buffer.Output_Table.Data[5].4);
   96: Cycle_Three_State(EditScenarioPv.Intrnl.AOI_Tg.RL_LP_B4_L2,EditScenario.Cmd.Trig_RL_LP_B4_L2,EditScenarioPv.Intrnl.Scenario_Edit_Buffer.Output_Table.Data[5].5,EditScenarioPv.Intrnl.Scenario_Edit_Buffer.Output_Table.Data[5].6);
   97: Cycle_Three_State(EditScenarioPv.Intrnl.AOI_Tg.RL_LP_B4_L3,EditScenario.Cmd.Trig_RL_LP_B4_L3,EditScenarioPv.Intrnl.Scenario_Edit_Buffer.Output_Table.Data[5].7,EditScenarioPv.Intrnl.Scenario_Edit_Buffer.Output_Table.Data[5].8);
   98: Cycle_Three_State(EditScenarioPv.Intrnl.AOI_Tg.RL_LP_B4_L4,EditScenario.Cmd.Trig_RL_LP_B4_L4,EditScenarioPv.Intrnl.Scenario_Edit_Buffer.Output_Table.Data[5].9,EditScenarioPv.Intrnl.Scenario_Edit_Buffer.Output_Table.Data[5].10);
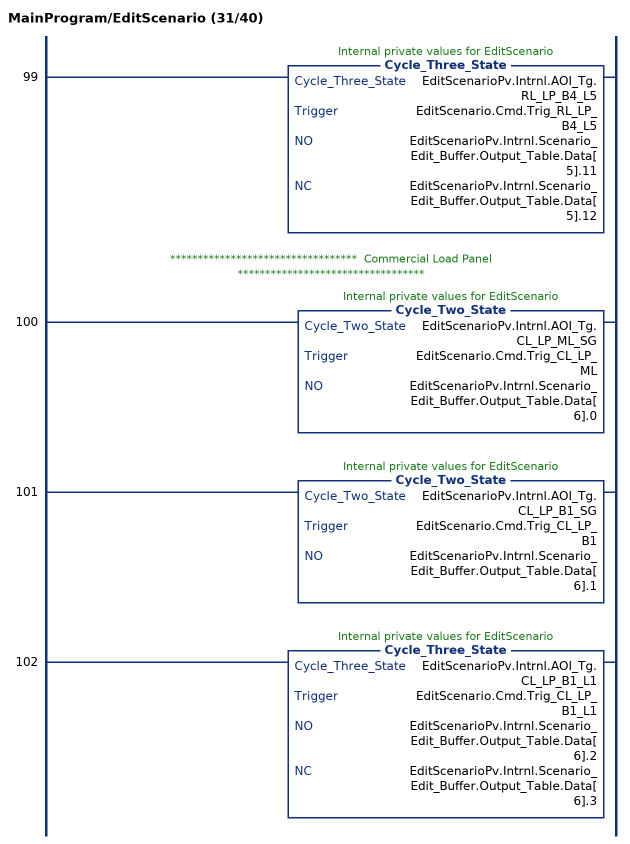
   99: Cycle_Three_State(EditScenarioPv.Intrnl.AOI_Tg.RL_LP_B4_L5,EditScenario.Cmd.Trig_RL_LP_B4_L5,EditScenarioPv.Intrnl.Scenario_Edit_Buffer.Output_Table.Data[5].11,EditScenarioPv.Intrnl.Scenario_Edit_Buffer.Output_Table.Data[5].12);
   // **********************************  Commercial Load Panel **********************************
   100: Cycle_Two_State(EditScenarioPv.Intrnl.AOI_Tg.CL_LP_ML_SG,EditScenario.Cmd.Trig_CL_LP_ML,EditScenarioPv.Intrnl.Scenario_Edit_Buffer.Output_Table.Data[6].0);
   101: Cycle_Two_State(EditScenarioPv.Intrnl.AOI_Tg.CL_LP_B1_SG,EditScenario.Cmd.Trig_CL_LP_B1,EditScenarioPv.Intrnl.Scenario_Edit_Buffer.Output_Table.Data[6].1);
   102: Cycle_Three_State(EditScenarioPv.Intrnl.AOI_Tg.CL_LP_B1_L1,EditScenario.Cmd.Trig_CL_LP_B1_L1,EditScenarioPv.Intrnl.Scenario_Edit_Buffer.Output_Table.Data[6].2,EditScenarioPv.Intrnl.Scenario_Edit_Buffer.Output_Table.Data[6].3);
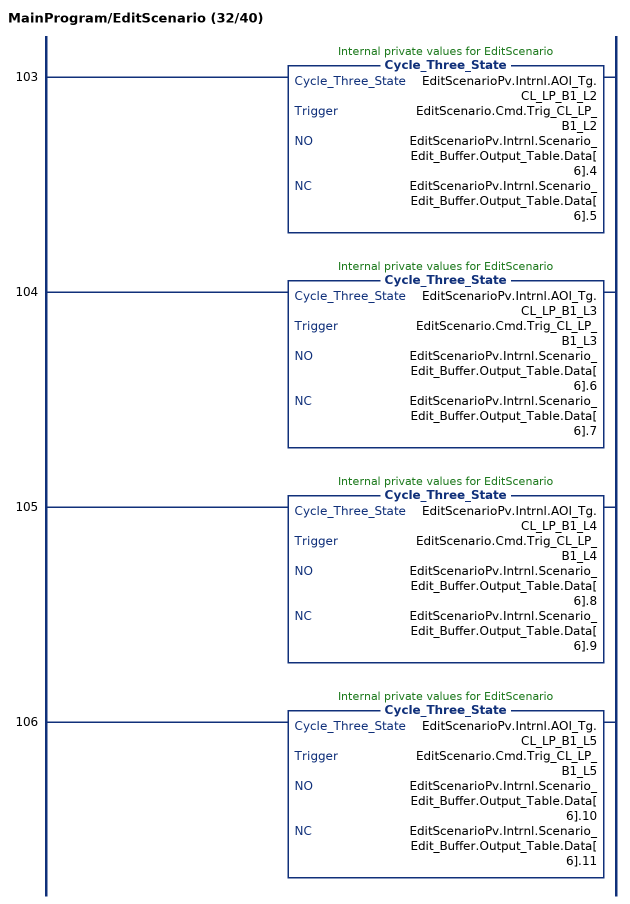
   103: Cycle_Three_State(EditScenarioPv.Intrnl.AOI_Tg.CL_LP_B1_L2,EditScenario.Cmd.Trig_CL_LP_B1_L2,EditScenarioPv.Intrnl.Scenario_Edit_Buffer.Output_Table.Data[6].4,EditScenarioPv.Intrnl.Scenario_Edit_Buffer.Output_Table.Data[6].5);
   104: Cycle_Three_State(EditScenarioPv.Intrnl.AOI_Tg.CL_LP_B1_L3,EditScenario.Cmd.Trig_CL_LP_B1_L3,EditScenarioPv.Intrnl.Scenario_Edit_Buffer.Output_Table.Data[6].6,EditScenarioPv.Intrnl.Scenario_Edit_Buffer.Output_Table.Data[6].7);
   105: Cycle_Three_State(EditScenarioPv.Intrnl.AOI_Tg.CL_LP_B1_L4,EditScenario.Cmd.Trig_CL_LP_B1_L4,EditScenarioPv.Intrnl.Scenario_Edit_Buffer.Output_Table.Data[6].8,EditScenarioPv.Intrnl.Scenario_Edit_Buffer.Output_Table.Data[6].9);
   106: Cycle_Three_State(EditScenarioPv.Intrnl.AOI_Tg.CL_LP_B1_L5,EditScenario.Cmd.Trig_CL_LP_B1_L5,EditScenarioPv.Intrnl.Scenario_Edit_Buffer.Output_Table.Data[6].10,EditScenarioPv.Intrnl.Scenario_Edit_Buffer.Output_Table.Data[6].11);
